# EPICS autosave request: iocBoot/ioc13bmd/auto_settings_xps.req
file "CARS_motor_settings.req",         P=$(P), M=m89
file "CARS_motor_settings.req",         P=$(P), M=m90
file "CARS_motor_settings.req",         P=$(P), M=m91
